// TIA Portal V19 export
DATA_BLOCK "A03_0102TrkManager"   // DB188
// stored: InstanceOfName A03_0102TrkManager_FB, InstanceOfType FB
"A03_0102TrkManager_FB"
   // VAR_INPUT
   //    AreaInterface : "AreaInterface";
   //    SuperUserLogged : Bool;
   // END_VAR
   // VAR
   //    HMI : Struct
   //       A0301_P : Struct
   //          Move : Array[1..11] of "TrkMng_Move";
   //       END_STRUCT;
   //       A0301_B : Struct
   //          Move : Array[1..12] of "TrkMng_Move";
   //       END_STRUCT;
   //       A0302_ENTRY : Struct
   //          Move : Array[1..7] of "TrkMng_Move";
   //       END_STRUCT;
   //       A0302_EXIT : Struct
   //          Move : Array[1..18] of "TrkMng_Move";
   //       END_STRUCT;
   //    END_STRUCT;
   //    Sts : Struct
   //       MoveA0301_P : Struct
   //          SelectionOn : Bool;
   //          SelectionNo : Int;
   //       END_STRUCT;
   //       MoveA0301_B : Struct
   //          SelectionOn : Bool;
   //          SelectionNo : Int;
   //       END_STRUCT;
   //       MoveA0302_ENTRY : Struct
   //          SelectionOn : Bool;
   //          SelectionNo : Int;
   //       END_STRUCT;
   //       MoveA0302_EXIT : Struct
   //          SelectionOn : Bool;
   //          SelectionNo : Int;
   //       END_STRUCT;
   //    END_STRUCT;
   //    A0301B_TON_Delete_Buttons : IEC_TIMER;
   //    A0301P_TON_Delete_Buttons : IEC_TIMER;
   //    A0302_ENTRY_TON_Delete_Buttons : IEC_TIMER;
   //    A0302_EXIT_TON_Delete_Buttons : IEC_TIMER;
   // END_VAR
BEGIN
END_DATA_BLOCK
